PROGRAM MAIN
VAR
END_VAR

(*Calling Different Programs*)
Motor_Control ();
ProgramSequence ();
Reset ();

END_PROGRAM

(* stored: Version 1.1.0.1, ProductVersion 3.1.4024.12
   POU MAIN: Id {17db34f9-79ec-460d-90c3-00845aea4c24}, SpecialFunc None *)
